// TIA Portal project "BTKetNoiFactoryIO&C#" (V18)

(* hardware
DEVICE "S7-1500/ET200MP station_1"  S7-1500 station
   slot 0: "Rail_0"  Rack  6ES7 590-1***0-0AA0
   slot 1: "PLC_1"  CPU 1513-1 PN  6ES7 513-1AL02-0AB0  V2.6
      slot 3: "CPU display_1"  6ES7591-1AA00-0AA0
      slot 32768: "PROFINET interface_1"  X1
         slot 32769: "Port_1"  X1 P1
         slot 32770: "Port_2"  X1 P2
   slot 2: "DI 16x24VDC BA_1"  DI 16x24VDC BA  6ES7 521-1BH10-0AA0  V1.1
   slot 3: "DQ 16x24VDC/0.5A BA_1"  DQ 16x24VDC/0.5A BA  6ES7 522-1BH10-0AA0  V1.1
*)

// ===== PLC "PLC_1"  CPU 1513-1 PN =====

VAR_GLOBAL   // PLC tag table "Default tag table"
   "System_Byte" AT %MB501 : Byte;
   "FirstScan" AT %M501.0 : Bool;
   "DiagStatusUpdate" AT %M501.1 : Bool;
   "AlwaysTRUE" AT %M501.2 : Bool;
   "AlwaysFALSE" AT %M501.3 : Bool;
   "Clock_Byte" AT %MB500 : Byte;
   "Clock_10Hz" AT %M500.0 : Bool;
   "Clock_5Hz" AT %M500.1 : Bool;
   "Clock_2.5Hz" AT %M500.2 : Bool;
   "Clock_2Hz" AT %M500.3 : Bool;
   "Clock_1.25Hz" AT %M500.4 : Bool;
   "Clock_1Hz" AT %M500.5 : Bool;
   "Clock_0.625Hz" AT %M500.6 : Bool;
   "Clock_0.5Hz" AT %M500.7 : Bool;
END_VAR

VAR_GLOBAL   // PLC tag table "Input"
   "Start" AT %I0.0 : Bool;
   "Stop" AT %I0.1 : Bool;
   "Reset" AT %I0.2 : Bool;
   "Sensor1" AT %I0.3 : Bool;
   "Sensor2" AT %I0.4 : Bool;
   "Sensor3" AT %I0.5 : Bool;
   "Sensor_CountC" AT %I0.6 : Bool;
   "Sensor_CountTB" AT %I0.7 : Bool;
   "Sensor_CountT" AT %I1.0 : Bool;
   "TurnFront" AT %I1.1 : Bool;
   "TurnBack" AT %I1.2 : Bool;
   "TurnLimit0" AT %I1.3 : Bool;
   "TurnLimit90" AT %I1.4 : Bool;
END_VAR

VAR_GLOBAL   // PLC tag table "Output"
   "Conveyor0" AT %Q0.0 : Bool;
   "Conveyor1" AT %Q0.1 : Bool;
   "Conveyor2" AT %Q0.2 : Bool;
   "Conveyor3" AT %Q0.3 : Bool;
   "TurnTableTurn" AT %Q0.4 : Bool;
   "TurnTableRoll+" AT %Q0.5 : Bool;
   "TurnTableRoll-" AT %Q0.6 : Bool;
   "Count_C" AT %QW30 : Int;
   "Count_TB" AT %QW32 : Int;
   "Count_T" AT %QW34 : Int;
END_VAR

VAR_GLOBAL   // PLC tag table "P_Table"
   "P1" AT %M50.0 : Bool;
   "P2" AT %M50.1 : Bool;
   "P3" AT %M50.2 : Bool;
   "P4" AT %M50.3 : Bool;
   "P5" AT %M50.4 : Bool;
   "P6" AT %M50.5 : Bool;
   "P7" AT %M50.6 : Bool;
   "P8" AT %M50.7 : Bool;
END_VAR

VAR_GLOBAL   // PLC tag table "TrungGian"
   "Run" AT %M0.0 : Bool;
   "StopC0" AT %M0.1 : Bool;
   "M_Start" AT %M0.2 : Bool;
   "M_Stop" AT %M0.3 : Bool;
   "M_Reset" AT %M0.4 : Bool;
END_VAR

DATA_BLOCK "DefinePlant_DB"   // DB1
{ S7_Optimized_Access := 'TRUE' }
VERSION : 0.1
// stored: InstanceOfName DefinePlant
"DefinePlant"
BEGIN
END_DATA_BLOCK

DATA_BLOCK "FB_Cao_DB"   // DB4
{ S7_Optimized_Access := 'TRUE' }
VERSION : 0.1
// stored: InstanceOfName FB_Cao
"FB_Cao"
BEGIN
END_DATA_BLOCK

DATA_BLOCK "FB_TrungBinh_DB"   // DB5
{ S7_Optimized_Access := 'TRUE' }
VERSION : 0.1
// stored: InstanceOfName FB_TrungBinh
"FB_TrungBinh"
BEGIN
END_DATA_BLOCK

DATA_BLOCK "FB_Ngan_DB"   // DB6
{ S7_Optimized_Access := 'TRUE' }
VERSION : 0.1
// stored: InstanceOfName FB_Ngan
"FB_Ngan"
BEGIN
END_DATA_BLOCK

// folder: System blocks/Program resources

DATA_BLOCK "IEC_Counter_0_DB"   // DB7
{ S7_Optimized_Access := 'TRUE' }
AUTHOR : Simatic
FAMILY : IEC
NAME : CNTR
VERSION : 1.0
// stored: InstanceOfName IEC_COUNTER
"IEC_COUNTER"
BEGIN
END_DATA_BLOCK

DATA_BLOCK "IEC_Counter_0_DB_1"   // DB8
{ S7_Optimized_Access := 'TRUE' }
AUTHOR : Simatic
FAMILY : IEC
NAME : CNTR
VERSION : 1.0
// stored: InstanceOfName IEC_COUNTER
"IEC_COUNTER"
BEGIN
END_DATA_BLOCK

DATA_BLOCK "IEC_Counter_0_DB_2"   // DB9
{ S7_Optimized_Access := 'TRUE' }
AUTHOR : Simatic
FAMILY : IEC
NAME : CNTR
VERSION : 1.0
// stored: InstanceOfName IEC_COUNTER
"IEC_COUNTER"
BEGIN
END_DATA_BLOCK

// folder: (top level)

FUNCTION_BLOCK "DefinePlant"   // FB1, LAD
{ S7_Optimized_Access := 'TRUE' }
VERSION : 0.1
   VAR_INPUT
      CB1 : Bool;
      CB2 : Bool;
      CB3 : Bool;
   END_VAR
   VAR_OUTPUT
      State : Int;
   END_VAR
   VAR_TEMP
      Cao : Bool;
      TrungBinh : Bool;
      Thap : Bool;
      P1 : Bool;
      P2 : Bool;
      P3 : Bool;
   END_VAR
   VAR_TEMP   // added for the SCL form of the ladder/FBD networks
      _w1 : Bool;
      _w2 : Bool;
      _w3 : Bool;
   END_VAR
BEGIN

REGION Network 1
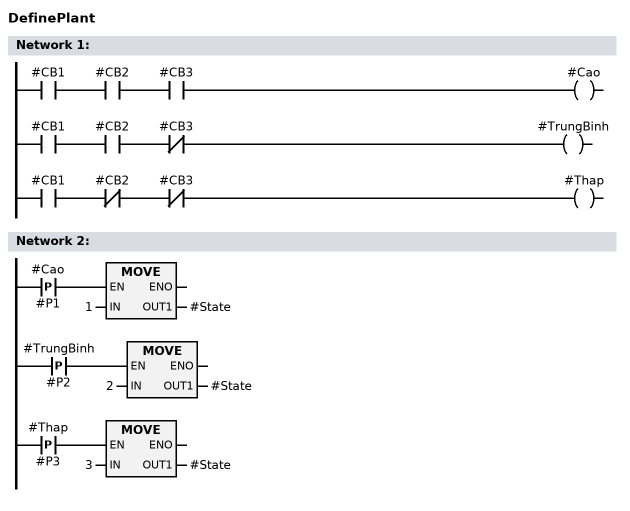
   RUNG wire#powerrail
      Contact( #CB1 )
      Contact( #CB2 )
      Contact( #CB3 )
      Coil( #Cao )
   END_RUNG
   RUNG wire#powerrail
      Contact( #CB1 )
      Contact( #CB2 )
      I_Contact( #CB3 )
      Coil( #TrungBinh )
   END_RUNG
   RUNG wire#powerrail
      Contact( #CB1 )
      I_Contact( #CB2 )
      I_Contact( #CB3 )
      Coil( #Thap )
   END_RUNG
   // the same network as SCL:
   #Cao := #CB1 AND #CB2 AND #CB3;
   #TrungBinh := #CB1 AND #CB2 AND NOT #CB3;
   #Thap := #CB1 AND NOT #CB2 AND NOT #CB3;
END_REGION

REGION Network 2
   RUNG wire#powerrail
      P_Contact(operand := #Cao, bit := #P1)
      Move(in := 1, out1 => #State)
   END_RUNG
   RUNG wire#powerrail
      P_Contact(operand := #TrungBinh, bit := #P2)
      Move(in := 2, out1 => #State)
   END_RUNG
   RUNG wire#powerrail
      P_Contact(operand := #Thap, bit := #P3)
      Move(in := 3, out1 => #State)
   END_RUNG
   // the same network as SCL:
   #_w1 := #Cao AND NOT #P1;   // rising edge of #Cao
   #P1 := #Cao;
   IF #_w1 THEN #State := 1; END_IF;
   #_w2 := #TrungBinh AND NOT #P2;   // rising edge of #TrungBinh
   #P2 := #TrungBinh;
   IF #_w2 THEN #State := 2; END_IF;
   #_w3 := #Thap AND NOT #P3;   // rising edge of #Thap
   #P3 := #Thap;
   IF #_w3 THEN #State := 3; END_IF;
END_REGION
END_FUNCTION_BLOCK

FUNCTION_BLOCK "FB_Cao"   // FB2, LAD
{ S7_Optimized_Access := 'TRUE' }
VERSION : 0.1
   VAR_OUTPUT
      Turn : Bool;
      "Roll+" : Bool;
      "Roll-" : Bool;
   END_VAR
BEGIN

REGION Network 1
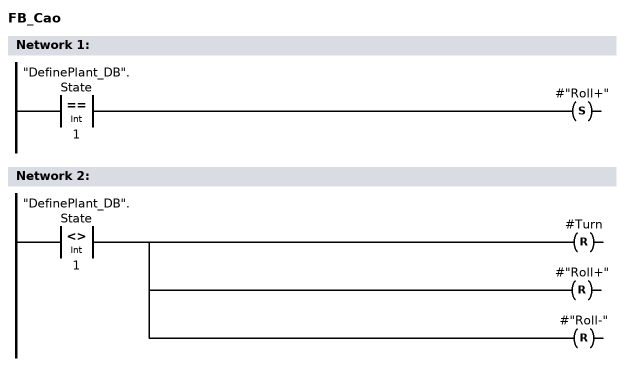
   RUNG wire#powerrail
      { S7_Templates := "SrcType := Int" } EQ_Contact(in1 := "DefinePlant_DB".State, in2 := 1)
      S_Coil( #"Roll+" )
   END_RUNG
   // the same network as SCL:
   IF "DefinePlant_DB".State = 1 THEN #"Roll+" := TRUE; END_IF;
END_REGION

REGION Network 2
   RUNG wire#powerrail
      { S7_Templates := "SrcType := Int" } NE_Contact(in1 := "DefinePlant_DB".State, in2 := 1)
      wire#w1
      R_Coil( #Turn )
   END_RUNG
   RUNG wire#w1
      R_Coil( #"Roll+" )
   END_RUNG
   RUNG wire#w1
      R_Coil( #"Roll-" )
   END_RUNG
   // the same network as SCL:
   IF "DefinePlant_DB".State <> 1 THEN
       #Turn := FALSE;
       #"Roll+" := FALSE;
       #"Roll-" := FALSE;
   END_IF;
END_REGION
END_FUNCTION_BLOCK

FUNCTION_BLOCK "FB_TrungBinh"   // FB3, LAD
{ S7_Optimized_Access := 'TRUE' }
VERSION : 0.1
   VAR_OUTPUT
      Turn : Bool;
      "Roll+" : Bool;
      "Roll-" : Bool;
   END_VAR
   VAR
      IEC_Timer_0_Instance : TON_TIME;
      IEC_Timer_0_Instance_1 : TON_TIME;
   END_VAR
   VAR_TEMP   // added for the SCL form of the ladder/FBD networks
      _w1 : Bool;
   END_VAR
BEGIN

REGION Network 1
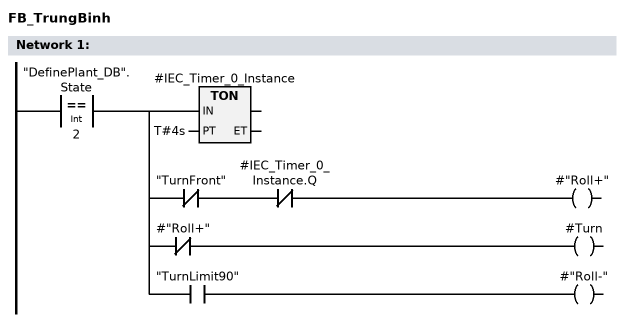
   #_w1 := "DefinePlant_DB".State = 2;
   #IEC_Timer_0_Instance(IN := #_w1, PT := T#4s);   // TON
   #"Roll+" := #_w1 AND NOT "TurnFront" AND NOT #IEC_Timer_0_Instance.Q;
   #Turn := #_w1 AND NOT #"Roll+";
   #"Roll-" := #_w1 AND "TurnLimit90";
END_REGION
END_FUNCTION_BLOCK

FUNCTION_BLOCK "FB_Ngan"   // FB4, LAD
{ S7_Optimized_Access := 'TRUE' }
VERSION : 0.1
   VAR_OUTPUT
      Turn : Bool;
      "Roll+" : Bool;
      "Roll-" : Bool;
   END_VAR
   VAR
      IEC_Timer_0_Instance : TON_TIME;
      temp : Bool;
   END_VAR
   VAR_TEMP   // added for the SCL form of the ladder/FBD networks
      _w1 : Bool;
   END_VAR
BEGIN

REGION Network 1
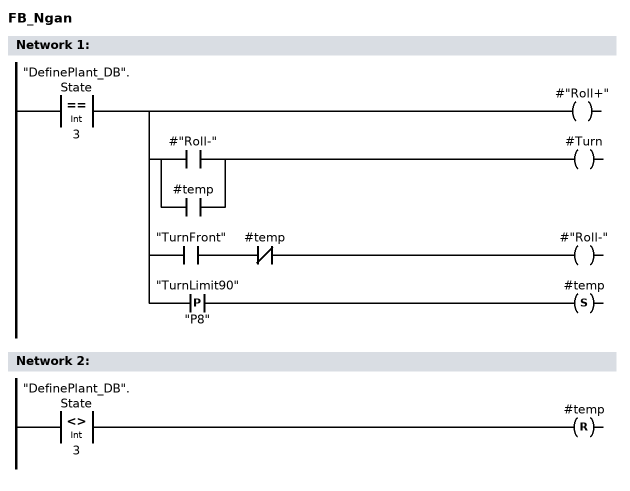
   RUNG wire#powerrail
      { S7_Templates := "SrcType := Int" } EQ_Contact(in1 := "DefinePlant_DB".State, in2 := 3)
      wire#w1
      Coil( #"Roll+" )
   END_RUNG
   RUNG wire#w1
      Contact( #"Roll-" )
      wire#w2
      Coil( #Turn )
   END_RUNG
   RUNG wire#w1
      Contact( #temp )
   END_RUNG wire#w2
   RUNG wire#w1
      Contact( "TurnFront" )
      I_Contact( #temp )
      Coil( #"Roll-" )
   END_RUNG
   RUNG wire#w1
      P_Contact(operand := "TurnLimit90", bit := "P8")
      S_Coil( #temp )
   END_RUNG
   // the same network as SCL:
   #"Roll+" := "DefinePlant_DB".State = 3;
   #Turn := #"Roll+" AND (#"Roll-" OR #temp);
   #"Roll-" := #"Roll+" AND "TurnFront" AND NOT #temp;
   #_w1 := #"Roll+" AND "TurnLimit90" AND NOT "P8";   // rising edge of "TurnLimit90"
   "P8" := "TurnLimit90";
   IF #_w1 THEN #temp := TRUE; END_IF;
END_REGION

REGION Network 2
   RUNG wire#powerrail
      { S7_Templates := "SrcType := Int" } NE_Contact(in1 := "DefinePlant_DB".State, in2 := 3)
      R_Coil( #temp )
   END_RUNG
   // the same network as SCL:
   IF "DefinePlant_DB".State <> 3 THEN #temp := FALSE; END_IF;
END_REGION
END_FUNCTION_BLOCK

ORGANIZATION_BLOCK "Main"   // OB1, LAD, ProgramCycle
TITLE = "Main Program Sweep (Cycle)"
{ S7_Optimized_Access := 'TRUE' }
VERSION : 0.1
   VAR_INPUT
      Initial_Call : Bool;   // Initial call of this OB
      Remanence : Bool;   // =True, if remanent data are available
   END_VAR
   VAR_TEMP   // added for the SCL form of the ladder/FBD networks
      _w1 : Bool;
      _w2 : Bool;
      _w3 : Bool;
   END_VAR
BEGIN

REGION Network 1
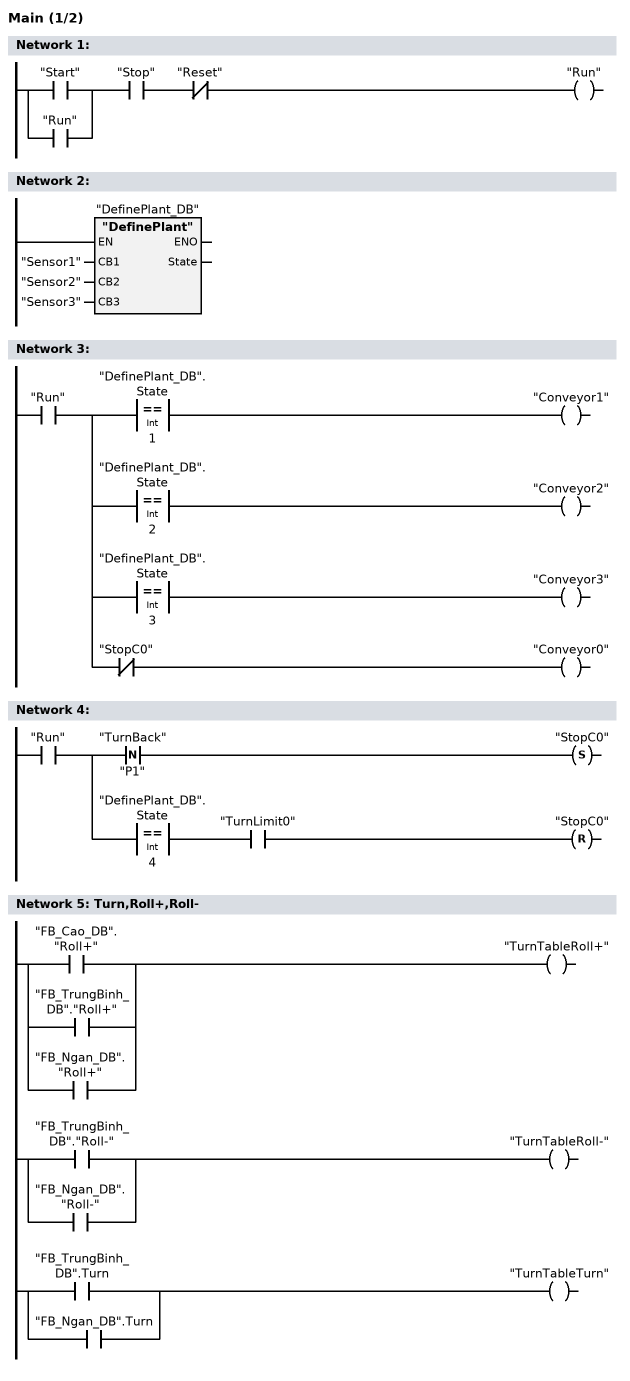
   RUNG wire#powerrail
      Contact( "Start" )
      wire#w1
      Contact( "Stop" )
      I_Contact( "Reset" )
      Coil( "Run" )
   END_RUNG
   RUNG wire#powerrail
      Contact( "Run" )
   END_RUNG wire#w1
   // the same network as SCL:
   "Run" := ("Start" OR "Run") AND "Stop" AND NOT "Reset";
END_REGION

REGION Network 2
   RUNG wire#powerrail
      "DefinePlant_DB"(CB1 := "Sensor1", CB2 := "Sensor2", CB3 := "Sensor3", State =>)
   END_RUNG
   // the same network as SCL:
   "DefinePlant_DB"(CB1 := "Sensor1", CB2 := "Sensor2", CB3 := "Sensor3");   // "DefinePlant"
END_REGION

REGION Network 3
   RUNG wire#powerrail
      Contact( "Run" )
      wire#w1
      { S7_Templates := "SrcType := Int" } EQ_Contact(in1 := "DefinePlant_DB".State, in2 := 1)
      Coil( "Conveyor1" )
   END_RUNG
   RUNG wire#w1
      { S7_Templates := "SrcType := Int" } EQ_Contact(in1 := "DefinePlant_DB".State, in2 := 2)
      Coil( "Conveyor2" )
   END_RUNG
   RUNG wire#w1
      { S7_Templates := "SrcType := Int" } EQ_Contact(in1 := "DefinePlant_DB".State, in2 := 3)
      Coil( "Conveyor3" )
   END_RUNG
   RUNG wire#w1
      I_Contact( "StopC0" )
      Coil( "Conveyor0" )
   END_RUNG
   // the same network as SCL:
   "Conveyor1" := "Run" AND ("DefinePlant_DB".State = 1);
   "Conveyor2" := "Run" AND ("DefinePlant_DB".State = 2);
   "Conveyor3" := "Run" AND ("DefinePlant_DB".State = 3);
   "Conveyor0" := "Run" AND NOT "StopC0";
END_REGION

REGION Network 4
   RUNG wire#powerrail
      Contact( "Run" )
      wire#w1
      N_Contact(operand := "TurnBack", bit := "P1")
      S_Coil( "StopC0" )
   END_RUNG
   RUNG wire#w1
      { S7_Templates := "SrcType := Int" } EQ_Contact(in1 := "DefinePlant_DB".State, in2 := 4)
      Contact( "TurnLimit0" )
      R_Coil( "StopC0" )
   END_RUNG
   // the same network as SCL:
   #_w1 := "Run" AND NOT "TurnBack" AND "P1";   // falling edge of "TurnBack"
   "P1" := "TurnBack";
   IF #_w1 THEN "StopC0" := TRUE; END_IF;
   IF "Run" AND ("DefinePlant_DB".State = 4) AND "TurnLimit0" THEN "StopC0" := FALSE; END_IF;
END_REGION

REGION Network 5: Turn,Roll+,Roll-
   RUNG wire#powerrail
      Contact( "FB_Cao_DB"."Roll+" )
      wire#w1
      Coil( "TurnTableRoll+" )
   END_RUNG
   RUNG wire#powerrail
      Contact( "FB_TrungBinh_DB"."Roll+" )
   END_RUNG wire#w1
   RUNG wire#powerrail
      Contact( "FB_Ngan_DB"."Roll+" )
   END_RUNG wire#w1
   RUNG wire#powerrail
      Contact( "FB_TrungBinh_DB"."Roll-" )
      wire#w2
      Coil( "TurnTableRoll-" )
   END_RUNG
   RUNG wire#powerrail
      Contact( "FB_Ngan_DB"."Roll-" )
   END_RUNG wire#w2
   RUNG wire#powerrail
      Contact( "FB_TrungBinh_DB".Turn )
      wire#w3
      Coil( "TurnTableTurn" )
   END_RUNG
   RUNG wire#powerrail
      Contact( "FB_Ngan_DB".Turn )
   END_RUNG wire#w3
   // the same network as SCL:
   "TurnTableRoll+" := "FB_Cao_DB"."Roll+" OR "FB_TrungBinh_DB"."Roll+" OR "FB_Ngan_DB"."Roll+";
   "TurnTableRoll-" := "FB_TrungBinh_DB"."Roll-" OR "FB_Ngan_DB"."Roll-";
   "TurnTableTurn" := "FB_TrungBinh_DB".Turn OR "FB_Ngan_DB".Turn;
END_REGION

REGION Network 6
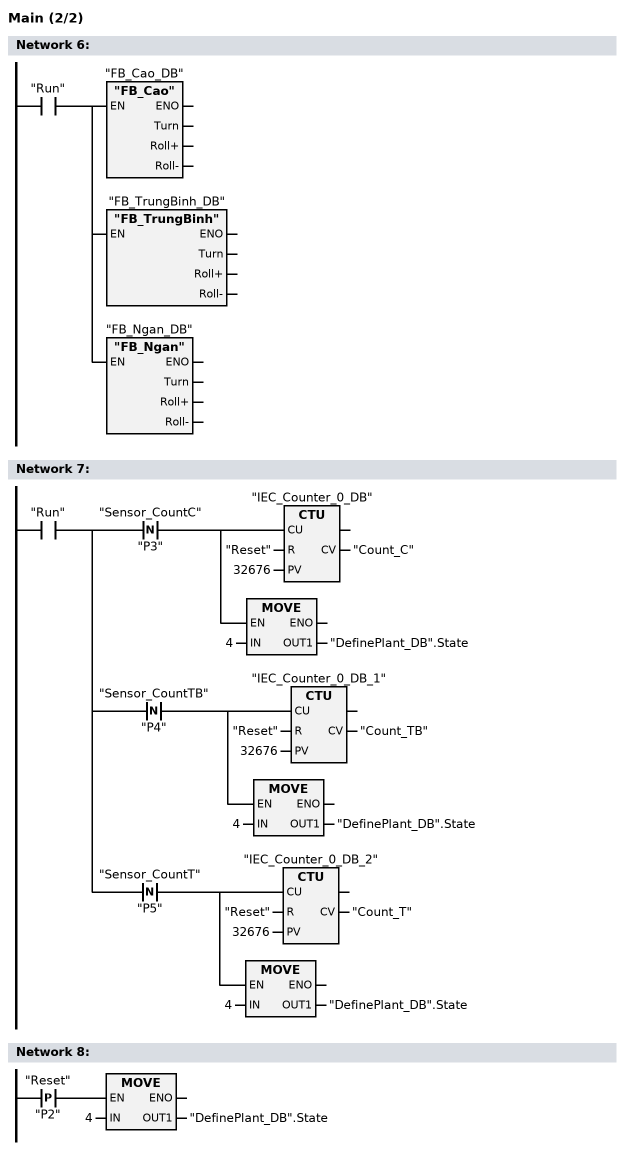
   RUNG wire#powerrail
      Contact( "Run" )
      wire#w1
      "FB_Cao_DB"(Turn =>, "Roll+" =>, "Roll-" =>)
   END_RUNG
   RUNG wire#w1
      "FB_TrungBinh_DB"(Turn =>, "Roll+" =>, "Roll-" =>)
   END_RUNG
   RUNG wire#w1
      "FB_Ngan_DB"(Turn =>, "Roll+" =>, "Roll-" =>)
   END_RUNG
   // the same network as SCL:
   #_w1 := "Run";
   IF #_w1 THEN
       "FB_Cao_DB"();   // "FB_Cao"
       "FB_TrungBinh_DB"();   // "FB_TrungBinh"
       "FB_Ngan_DB"();   // "FB_Ngan"
   END_IF;
END_REGION

REGION Network 7
   #_w1 := "Run" AND NOT "Sensor_CountC" AND "P3";   // falling edge of "Sensor_CountC"
   "P3" := "Sensor_CountC";
   "IEC_Counter_0_DB".CTU(CU := #_w1, R := "Reset", PV := 32676, CV => "Count_C");
   IF #_w1 THEN "DefinePlant_DB".State := 4; END_IF;
   #_w2 := "Run" AND NOT "Sensor_CountTB" AND "P4";   // falling edge of "Sensor_CountTB"
   "P4" := "Sensor_CountTB";
   "IEC_Counter_0_DB_1".CTU(CU := #_w2, R := "Reset", PV := 32676, CV => "Count_TB");
   IF #_w2 THEN "DefinePlant_DB".State := 4; END_IF;
   #_w3 := "Run" AND NOT "Sensor_CountT" AND "P5";   // falling edge of "Sensor_CountT"
   "P5" := "Sensor_CountT";
   "IEC_Counter_0_DB_2".CTU(CU := #_w3, R := "Reset", PV := 32676, CV => "Count_T");
   IF #_w3 THEN "DefinePlant_DB".State := 4; END_IF;
END_REGION

REGION Network 8
   RUNG wire#powerrail
      P_Contact(operand := "Reset", bit := "P2")
      Move(in := 4, out1 => "DefinePlant_DB".State)
   END_RUNG
   // the same network as SCL:
   #_w1 := "Reset" AND NOT "P2";   // rising edge of "Reset"
   "P2" := "Reset";
   IF #_w1 THEN "DefinePlant_DB".State := 4; END_IF;
END_REGION
END_ORGANIZATION_BLOCK